{attribute 'reflection'}
FUNCTION_BLOCK ABSTRACT Label IMPLEMENTS I_Label
VAR CONSTANT
END_VAR
VAR_INPUT
END_VAR
VAR
	
	{attribute 'instance-path'} 
    {attribute 'noinit'}
	_sPath: T_MaxString;
	{attribute 'no_copy'}
	_name: T_MaxString;
	
END_VAR

//Base class. Allows to querry instances by their name.

METHOD FB_init : BOOL
VAR_INPUT
	bInitRetains : BOOL; // if TRUE, the retain variables are initialized (warm start / cold start)
	bInCopyCode : BOOL;  // if TRUE, the instance afterwards gets moved into the copy code (online change)
END_VAR
//Update name after each 'New Download'
_name := DELETE(_sPath, FIND(_sPath, '.'), 1);
_name := DELETE(_name, FIND(_name, '.'), 1);
END_METHOD

PROPERTY name : STRING
GET
name := _name;
END_GET
END_PROPERTY

END_FUNCTION_BLOCK

(* stored: Version 1.1.0.1, ProductVersion 3.1.4024.12
   POU Label: Id {1ca27162-a753-4627-9fe0-11386270227f}, SpecialFunc None
   Method FB_init: Id {2fdf334e-2b2d-4639-ba14-26a06891310e}
   Property name: Id {51ac3072-3c91-47be-8c6f-4ddd0aa84d6c}
   Get Get: Id {434a7f2a-0410-41bd-a9ea-abda52936d77} *)
